FUNCTION_BLOCK LString
VAR_INPUT
END_VAR
VAR_OUTPUT
END_VAR
VAR
  _str: STRING(255);
  _length: INT;
END_VAR

METHOD PUBLIC append
VAR_IN_OUT
  lstr: LString; 
END_VAR
MEMMOVE(
  destAddr:=ADR(_str)+TO_DWORD(length),
  srcAddr:=ADR(lstr._str),
  n:=TO_UDINT(lstr.length+1));
length := length + lstr.length;
END_METHOD

METHOD PUBLIC append_str
VAR_INPUT
  str: STRING(255);
END_VAR
VAR
  length: INT;
END_VAR
length := LEN(str);
MEMMOVE(
  destAddr:=ADR(_str)+TO_DWORD(THIS^.length),
  srcAddr:=ADR(str),
  n:=TO_UDINT(length+1));
THIS^.length := THIS^.length + length;
END_METHOD

PROPERTY PUBLIC length : INT
GET
length := _length;
END_GET
SET // PRIVATE
_length := length;
END_SET
END_PROPERTY

METHOD PUBLIC remove_left_including_char
VAR_INPUT
  char: STRING(1);
  number: INT;
END_VAR
VAR
  act_number: INT;
  offset: INT;
  i: INT;
END_VAR
WHILE _str[i] <> 0 DO
  IF act_number < number THEN
    IF _str[i] = char[0] THEN
      act_number := act_number + 1;
    END_IF
  ELSE
    EXIT;
	END_IF
  i := i + 1;
END_WHILE
MEMMOVE(
  destAddr:=ADR(_str),
  srcAddr:=ADR(_str)+TO_DWORD(i),
  n:=TO_UDINT(length-i));
length := length - i;
_str[length] := 0;
END_METHOD

PROPERTY PUBLIC str : STRING(255)
GET
str := _str;
END_GET
SET
_str := str;
length := LEN(str);
END_SET
END_PROPERTY

END_FUNCTION_BLOCK

(* stored: Version 1.1.0.1, ProductVersion 3.1.4024.9
   POU LString: Id {33f4feb9-6553-4430-ac72-271fe5fcf8e4}, SpecialFunc None
   Method append: Id {eee8c8db-46af-4231-bc5d-9c51482a2cbf}
   Method append_str: Id {4e1327c3-c229-44c0-af49-8b9a41f66505}
   Property length: Id {59958980-3dda-4623-84b3-a87c55c1c2a2}
   Get Get: Id {8e8132ec-7a67-4a76-8600-1e35cc405b75}
   Set Set: Id {7399b23d-69cf-4ad9-b49c-51afbe8a7fb8}
   Method remove_left_including_char: Id {968542c2-bcb2-4f71-974c-51d0564fbae4}
   Property str: Id {cb130ec0-9141-44e1-b370-410dc6ceaaf1}
   Get Get: Id {bf8ac549-5821-480a-966e-cb0bab4c54f7}
   Set Set: Id {77e65917-d278-4fd9-a51a-7a8dfab88016} *)
